(* IEC 61131-3 sources: LASAL/Class/RefSwitchCurrent, 1 file *)

(* ---- RefSwitchCurrent.st ---- *)
(*!
<Class
	Name               = "RefSwitchCurrent"
	Revision           = "0.0"
	RealtimeTask       = "true"
	DefRealtime        = "1 ms"
	CyclicTask         = "false"
	BackgroundTask     = "false"
	Sigmatek           = "false"
	OSInterface        = "false"
	HighPriority       = "false"
	Automatic          = "false"
	UpdateMode         = "Prescan"
	SharedCommandTable = "true"
	Objectsize         = "(284,120)">
	<Channels>
		<Server Name="setpoint" Visualized="false" Initialize="true" WriteProtected="false" Retentive="File"/>
		<Server Name="Switch" Visualized="false" Initialize="false" WriteProtected="true" Retentive="false"/>
		<Client Name="Current" Required="true" Internal="false"/>
	</Channels>
</Class>
*)
RefSwitchCurrent : CLASS
  //Servers:
	setpoint 	: SvrChCmd_DINT;
	Switch 	: SvrCh_DINT;
  //Clients:
	Current 	: CltCh_DINT;
  //Variables:
  //Functions:

	FUNCTION VIRTUAL GLOBAL RtWork
		VAR_INPUT
			EAX 	: UDINT;
		END_VAR
		VAR_OUTPUT
			state (EAX) 	: UDINT;
		END_VAR;
  //Tables:
	FUNCTION @STD
		VAR_OUTPUT
			ret_code	: CONFSTATES;
		END_VAR;
	FUNCTION GLOBAL TAB @CT_;
END_CLASS;

FUNCTION VIRTUAL GLOBAL RefSwitchCurrent::RtWork
	VAR_INPUT
		EAX 	: UDINT;
	END_VAR
	VAR_OUTPUT
		state (EAX) 	: UDINT;
	END_VAR

  Current:=Current.Read();
  Switch:=abs(Current)>setpoint;

  state := READY;

END_FUNCTION
